// TIA Portal V20 export
DATA_BLOCK "BK07"   // DB202
// stored: MemoryReserve 100
   VAR
      "X10-1 POSITION MOVING LIMIT SENSOR(-)" : Bool;
      "X11-1 POSITION MOVING LIMIT SENSOR(+)" : Bool;
      "X12-1 VISION HOMING SENSOR" : Bool;
      "X13-1 ELECTRODE NG KICKER HOMING SENSOR" : Bool;
      "X14-1 ELECTRODE NG BOX FULL SENSOR" : Bool;
      "X15-1 ELECTRODE NG BOX DETECT SENSOR" : Bool;
      "X16-1 NG & MANUAL INPUT MAGAZINE FULL SENSOR" : Bool;
      "X17-1 MAGAZINE Z-AXIS SAFETY PIN POSITION SENSOR" : Bool;
      "X10-2 POSITION MOVING HOMING SENSOR" : Bool;
      "X11-2 CUTTER HOMING SENSOR" : Bool;
      "X12-2 SPARE" : Bool;
      "X13-2 ELECTRODE PASS KICKER HOMING SENSOR" : Bool;
      "X14-2 SPARE" : Bool;
      "X15-2 SPARE" : Bool;
      "X16-2 SPARE" : Bool;
      "X17-2 SPARE" : Bool;
   END_VAR
BEGIN
END_DATA_BLOCK
